// TwinCAT 3 PLC project CX5240
// ProgramVersion: 3.1.4026.13
// CompilerDefines: VISU_USEPROPERTYINFO
// libraries:
//   CmpBitmapPool, * (System)
//   Tc2_Standard, * (Beckhoff Automation GmbH)
//   Tc2_System, * (Beckhoff Automation GmbH)
//   Tc3_Module, * (Beckhoff Automation GmbH)
//   VisuDialogs, * (System)
//   VisuSymbols,3.5.10.0,System
// project tree:
//   Enums/ E_Status.TcDUT (not stored)
//   Function Blocks/ FB_AnalogInputScaling.TcPOU (not stored), FB_DisplacementControl.TcPOU (not stored), FB_Encoder.TcPOU (not stored), FB_Integrator.TcPOU (not stored), FB_Joystick.TcPOU (not stored), FB_JoystickInputScaling.TcPOU (not stored), FB_DisplacementValveOutput.TcPOU (not stored), FB_StartPos.TcPOU (not stored), FB_YokeInputScaling.TcPOU (not stored), FB_ValveOutput.TcPOU (not stored)
//   / GlobalTextList.TcGTLO, HMI.TcVIS, PlcTask.TcTTO (not stored), Visualization Manager.TcVMO (not stored)
//   GVLs/ G_IO.TcGVL, G_Parameters.TcGVL, G_Sensors.TcGVL (not stored), HMI.TcGVL
//   POUs/ MAIN.TcPOU (not stored), P_Inputs.TcPOU, P_MotionControl.TcPOU, P_Outputs.TcPOU (not stored)
//   Struct/ ST_AnalogInputScaling.TcDUT (not stored), ST_JoystickInputScaling.TcDUT (not stored), ST_YokeInputScaling.TcDUT (not stored), ST_Parameters.TcDUT (not stored), ST_ValveDeadBand.TcDUT (not stored), ST_ValveOutput.TcDUT (not stored)
// real-time tasks:
//   TASK PlcTask: cycle T#1ms, priority 20, ADS port 350
// I/O:
//   DEVICE Device 1 (EtherCAT), AmsNetId 128.39.200.126.2.1
//     Term 1 (EK1200) [EK1200-5000 EtherCAT Power supply (2A E-Bus)]
//       Term 2 (EL1859) [EL1859 8Ch. Dig. Input 24V, 3ms, 8Ch. Dig. Output 24V, 0.5A]
//       Term 3 (EL3174) [EL3174 4Ch. Ana. Input +/-10V Diff., +/-20mA SingleEnded, 16 Bit]
//       Term 4 (EL4032) [EL4032 2Ch. Ana. Output +/-10V, 12bit]
//       Term 7 (EL3204) [EL3204 4Ch. Ana. Input PT100 (RTD)]
//       Term 8 (EK1110) [EK1110 EtherCAT extension]
//     Term 14 (EK1818) [EK1818 EtherCAT IO-Coupler  (1A E-Bus, 8 Ch. Dig. In, 3ms, 4 Ch. Dig. Out 24V, 0,5A)]
//       Term 10 (EL1008) [EL1008 8Ch. Dig. Input 24V, 3ms]
//       Term 11 (EL3174) [EL3174 4Ch. Ana. Input +/-10V Diff., +/-20mA SingleEnded, 16 Bit]
//       Term 12 (EL3068) [EL3068 8Ch. Ana. Input 0-10V]
//       Term 5 (EL4032) [EL4032 2Ch. Ana. Output +/-10V, 12bit]
//       Term 6 (EL4122) [EL4122 2Ch. Ana. Output  4-20mA, 16bit]
//       Term 17 (EL9011) [EL9011 End Terminal]
//     Box 13 (Fraba EtherCAT) [Absolute Rotary Encoder IXARC V01.05]
// variable links:
//   CX5240/CX5240 Instance <-> Device 1 (EtherCAT)/Term 1 (EK1200)/Term 2 (EL1859)
//     PlcTask Inputs/G_IO.bTestNew <-> Channel 1/Input
//     PlcTask Outputs/G_IO.OutTestNew <-> Channel 9/Output
//   CX5240/CX5240 Instance <-> Device 1 (EtherCAT)/Term 1 (EK1200)/Term 3 (EL3174)
//     PlcTask Inputs/G_IO.nTestNew <-> AI Standard Channel 1/Value
//   CX5240/CX5240 Instance <-> Device 1 (EtherCAT)/Term 14 (EK1818)
//     PlcTask Inputs/G_IO.bEmgOk <-> Channel 1/Input
//     PlcTask Outputs/G_IO.bEnablePCDV <-> Channel 10/Output
//     PlcTask Outputs/G_IO.bOpenBrakes <-> Channel 9/Output
//     PlcTask Outputs/G_IO.bWinchValveEnable <-> Channel 11/Output
//   CX5240/CX5240 Instance <-> Device 1 (EtherCAT)/Term 14 (EK1818)/Term 10 (EL1008)
//     PlcTask Inputs/G_IO.bAutoSwtich <-> Channel 3/Input
//     PlcTask Inputs/G_IO.bDisplacementEnable <-> Channel 7/Input
//     PlcTask Inputs/G_IO.bManualSwtich <-> Channel 1/Input
//     PlcTask Inputs/G_IO.bOffSwtich <-> Channel 2/Input
//     PlcTask Inputs/G_IO.bStartButton <-> Channel 4/Input
//     PlcTask Inputs/G_IO.bStopButton <-> Channel 5/Input
//     PlcTask Inputs/G_IO.bWinchEnable <-> Channel 6/Input
//   CX5240/CX5240 Instance <-> Device 1 (EtherCAT)/Term 14 (EK1818)/Term 11 (EL3174)
//     PlcTask Inputs/G_IO.fPDCVMonitor <-> AI Standard Channel 1/Value
//     PlcTask Inputs/G_IO.fYoke <-> AI Standard Channel 4/Value
//     PlcTask Inputs/G_IO.nMoogMonitor <-> AI Standard Channel 2/Value
//   CX5240/CX5240 Instance <-> Device 1 (EtherCAT)/Term 14 (EK1818)/Term 12 (EL3068)
//     PlcTask Inputs/G_IO.fJoyXraw <-> AI Standard Channel 6/Value
//     PlcTask Inputs/G_IO.fJoyYraw <-> AI Standard Channel 7/Value
//     PlcTask Inputs/G_IO.fJoyZraw <-> AI Standard Channel 8/Value
//     PlcTask Inputs/G_IO.fPressureReturn <-> AI Standard Channel 3/Value
//     PlcTask Inputs/G_IO.fPressureSupply <-> AI Standard Channel 2/Value
//     PlcTask Inputs/G_IO.fPressureWinchA <-> AI Standard Channel 1/Value
//     PlcTask Inputs/G_IO.fPressureWinchB <-> AI Standard Channel 4/Value
//   CX5240/CX5240 Instance <-> Device 1 (EtherCAT)/Term 14 (EK1818)/Term 5 (EL4032)
//     PlcTask Outputs/G_IO.fWinchPDCVOut <-> AO Outputs Channel 1/Analog output
//   CX5240/CX5240 Instance <-> Device 1 (EtherCAT)/Term 14 (EK1818)/Term 6 (EL4122)
//     PlcTask Outputs/G_IO.fWinchValveOut <-> Channel 1/Output

// ---- GVLs/G_IO.TcGVL
{attribute 'qualified_only'}
VAR_GLOBAL
	// Digital Inputs
	bEmgOk 			     AT %I* : BOOL; 
	bStartButton 	     AT %I* : BOOL;
	bStopButton 	     AT %I* : BOOL; 
	bOffSwtich		     AT %I* : BOOL;  
	bManualSwtich	     AT %I* : BOOL; 
	bAutoSwtich			 AT %I* : BOOL; 
	bWinchEnable 		 AT %I* : BOOL; 
	bDisplacementEnable  AT %I* : BOOL;
	
	// Analog Intputs
	fJoyXraw 			 AT %I* : INT; 
	fJoyYraw			 AT %I* : INT; 
	fJoyZraw 			 AT %I* : INT; 
	fPDCVMonitor		 AT %I* : INT; 
	nMoogMonitor		 AT %I* : INT; 
	fYoke				 AT %I* : INT; 
	fPressureWinchA 	 AT %I* : INT; 
	fPressureWinchB 	 AT %I* : INT; 
	fPressureSupply 	 AT %I* : INT; 
	fPressureReturn 	 AT %I* : INT; 
	nWinchEncoderValue	 AT %I* : UDINT; 
	
	// Digital Outputs
	bOpenBrakes 		 AT %Q* : BOOL; 
	bEnablePCDV 		 AT %Q* : BOOL; 
	bWinchValveEnable 	 AT %Q* : BOOL; 
	
	// Analog Outputs
	fWinchPDCVOut 		 AT %Q* : INT := 10000; 
	fWinchValveOut 		 AT %Q* : INT := 16383; 
	
	// New Test
	bTestNew AT %I* : BOOL;
	nTestNew AT %I* : INT;
	
END_VAR

// ---- GVLs/G_Parameters.TcGVL
{attribute 'qualified_only'}
VAR_GLOBAL
stParam : ST_Parameters;
END_VAR

// ---- GVLs/HMI.TcGVL
{attribute 'qualified_only'}
VAR_GLOBAL
	bEndStopOverride : BOOL; 
	fTest			 : LREAL;
END_VAR

// ---- POUs/P_Inputs.TcPOU
PROGRAM P_Inputs
VAR
	fbJoystickWinch 				: FB_JoystickInputScaling;
	fbJoystickRot 					: FB_JoystickInputScaling;
	fbYokeInputScaling 				: FB_YokeInputScaling;
	fbWinchPosition 				: FB_Encoder;
	fbPressureSupply 				: FB_AnalogInputScaling;
	fbPressureReturn 				: FB_AnalogInputScaling;
	fbPressureWinch_A_Input 		: FB_AnalogInputScaling;
	fbPressureWinch_B_Output		: FB_AnalogInputScaling;
END_VAR

fbJoystickWinch(
	bEnable := G_IO.bManualSwtich OR G_IO.bAutoSwtich,
	nRawInput := G_IO.fJoyYraw,
	stJoystickInputScaling := G_Parameters.stParam.stJoystickInputScalingY,
	fNormalizedOutput => G_Sensors.fJoystickNormalizedY
);

fbJoystickRot(
	bEnable := G_IO.bManualSwtich,
	nRawInput := G_IO.fJoyZraw,
	stJoystickInputScaling := G_Parameters.stParam.stJoystickInputScalingZ,
	fNormalizedOutput => G_Sensors.fJoystickNormalizedZ
);

fbYokeInputScaling(
	bEnable := G_IO.bManualSwtich,
	nRawInput := G_IO.fYoke,
	stYokeInputScaling := G_Parameters.stParam.stYokeInputScaling,
	fNormalizedOutput => G_Sensors.fYokeNormalizedFeedback
);

fbWinchPosition (
	nRawInput := G_IO.nWinchEncoderValue, 
	fEncoderOffset := G_Parameters.stParam.fWinchEncoderOffset,
	fPosition => G_Sensors.fWinchEncoderPosition
);

fbPressureSupply(
	nRawInput := G_IO.fPressureSupply,
	stAnalogInputScaling := G_Parameters.stParam.stPressureSensorScaling400bar,
	fOutput => G_Sensors.fPressureSupply
);

fbPressureReturn(
	nRawInput := G_IO.fPressureReturn,
	stAnalogInputScaling := G_Parameters.stParam.stPressureSensorScaling40bar,
	fOutput => G_Sensors.fPressureReturn
);

fbPressureWinch_A_Input(
	nRawInput := G_IO.fPressureWinchA,
	stAnalogInputScaling := G_Parameters.stParam.stPressureSensorScaling400bar,
	fOutput => G_Sensors.fPressureWinchA
);

fbPressureWinch_B_Output(
	nRawInput := G_IO.fPressureCylinderA,
	stAnalogInputScaling := G_Parameters.stParam.stPressureSensorScaling400bar,
	fOutput => G_Sensors.fPressureWinchB
);

G_Sensors.fDeltaPMotor := (G_Sensors.fPressureWinchB - G_Sensors.fPressureWinchA);

END_PROGRAM

// ---- POUs/P_MotionControl.TcPOU
PROGRAM P_MotionControl
VAR
	fbJoystick 				: FB_Joystick;
	fbGetStartPos 			: FB_StartPos;
	fbWinchVelIntegrator 	: FB_Integrator;
	fWinchVelRef 			: LREAL;
	fWinchPosRef 			: LREAL;
	fWinchPos 				: LREAL;
	fInitialWinchPos 		: LREAL;
	bWinchVelIntegratorOn	: BOOL := TRUE; 
	bAutoEnable 			: BOOL;
	bManualEnable 			: BOOL;
	fWinchPosRefManual 		: LREAL;
	fWinchVelRefManual 		: LREAL;
	fWinchVelRefAuto 		: LREAL;
	fbJoyTest 				: FB_Joystick;
END_VAR

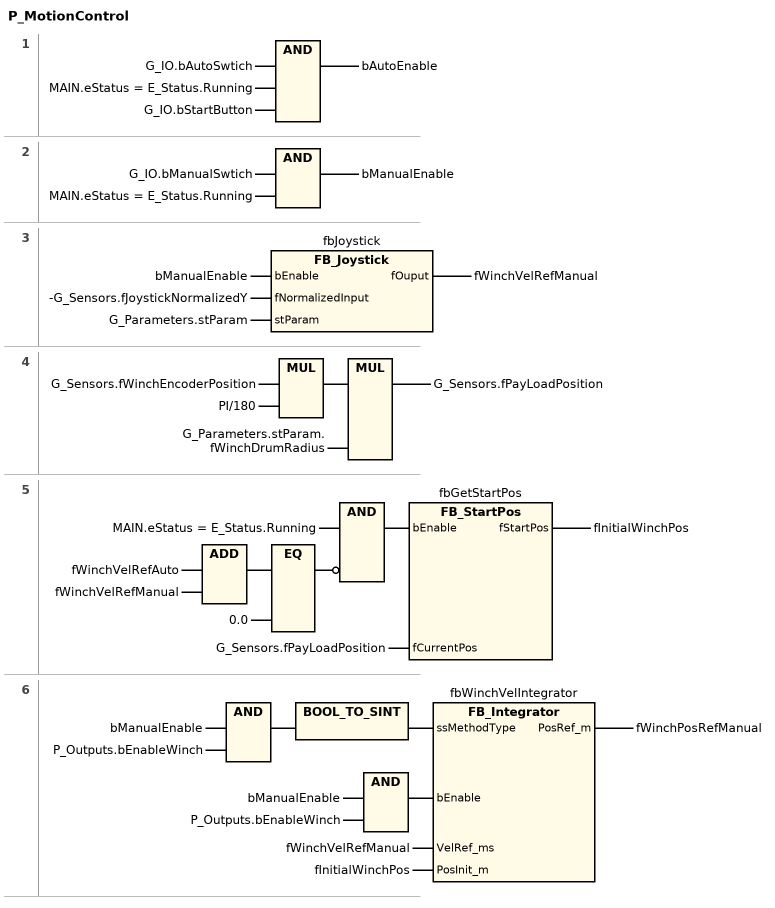
// NETWORK 1
bAutoEnable := G_IO.bAutoSwtich AND (MAIN.eStatus = E_Status.Running) AND G_IO.bStartButton;

// NETWORK 2
bManualEnable := G_IO.bManualSwtich AND (MAIN.eStatus = E_Status.Running);

// NETWORK 3
fbJoystick(
    bEnable := bManualEnable,
    fNormalizedInput := -G_Sensors.fJoystickNormalizedY,
    stParam := G_Parameters.stParam); // FB_Joystick
fWinchVelRefManual := fbJoystick.fOuput;

// NETWORK 4
G_Sensors.fPayLoadPosition := (G_Sensors.fWinchEncoderPosition * (PI/180)) * G_Parameters.stParam.fWinchDrumRadius;

// NETWORK 5
fbGetStartPos(bEnable := (MAIN.eStatus = E_Status.Running) AND NOT (fWinchVelRefAuto + fWinchVelRefManual = 0.0), fCurrentPos := G_Sensors.fPayLoadPosition); // FB_StartPos
fInitialWinchPos := fbGetStartPos.fStartPos;

// NETWORK 6
fbWinchVelIntegrator(
    ssMethodType := BOOL_TO_SINT(bManualEnable AND P_Outputs.bEnableWinch),
    bEnable := bManualEnable AND P_Outputs.bEnableWinch,
    VelRef_ms := fWinchVelRefManual,
    PosInit_m := fInitialWinchPos); // FB_Integrator
fWinchPosRefManual := fbWinchVelIntegrator.PosRef_m;

END_PROGRAM

// ---- GlobalTextList.TcGTLO
TEXTLIST GlobalTextList
  455 = '%2.1f'
  509 = '%2.2f'
  108 = '%f'
  308 = '%i'
  805 = '%I'
  528 = "'amplitude"
  341 = 'A'
  810 = 'Actvting Log P'
  221 = 'Actvting Log Plat'
  505 = 'Actvting Log Pos'
  560 = 'Amplitud'
  159 = 'Amplitude'
  639 = 'bar'
  175 = 'Controlelr'
  786 = 'Controller'
  847 = 'D'
  489 = 'END STOP OVERRIDE'
  897 = 'END STOP OVERRIDE '
  616 = 'EndStop Override'
  141 = 'GO TO SETTINGS'
  499 = 'I'
  490 = 'Main'
  911 = 'Main Screen'
  508 = 'Motion Control'
  934 = 'MOTION LIMIT'
  673 = 'Motion Limit'
  176 = 'MOTION LIMIT: OFF'
  449 = 'MOTION LIMITATION'
  802 = 'MOTION LIMITATION: OFF'
  69 = 'Neg End Stop'
  444 = 'Neg EndStop'
  896 = 'OVERRIDE'
  993 = 'P'
  312 = 'PA bar'
  288 = 'PA Winch bar'
  641 = 'PB bar'
  622 = 'PI COntroler'
  326 = 'PI Controler'
  878 = 'PI Displacement Control'
  623 = 'PI Gain DC'
  962 = 'PI Gain P'
  177 = 'PI Gain SC'
  28 = 'PI Primary Control'
  144 = 'PI Secondary Control'
  68 = 'PID'
  907 = 'PID Contoler'
  714 = 'PID Controller'
  706 = 'Pos End Stop'
  398 = 'Pos EndStop'
  309 = 'Position Logging'
  953 = 'Screen'
  358 = 'Secondary Control'
  699 = 'Secondry'
  663 = 'Secondry  swicher Primery'
  725 = 'Secondry Control'
  395 = 'Secondry Ish'
  17 = 'Secondry Swicher Primery'
  238 = 'Setings'
  169 = 'Settings'
  590 = 'Sin AmplitudContoler'
  156 = 'Sin TimeP Contoler'
  94 = 'Sin Wave'
  613 = 'Sin Wave Contoler'
  420 = 'Sine Motion Off/On'
  636 = 'Sine Wave'
  818 = 'Start Mual'
  898 = 'Time'
  26 = 'Time P'
  140 = 'Time Periode [s]'
  844 = 'TimeP'
  826 = 'TimePTime'
  402 = 'to Main'
  655 = 'Togel Swich Motion Control'
  469 = 'TURN ON IN SETTINGS'
  191 = 'Visualisation'
  345 = 'Visualiztion'
  718 = 'WARNING'
  113 = 'Warning ON'
  628 = 'Wave Amplitude [m]'
  592 = 'Working Progres'
  500 = 'XXX'
END_TEXTLIST

// ---- HMI.TcVIS
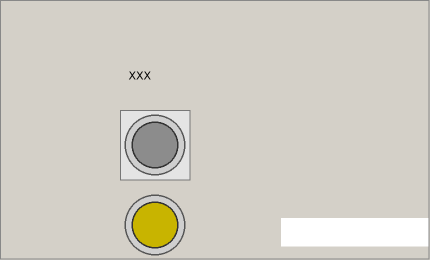
VISUALIZATION HMI  // 430x260
    PushSwitch (120,110 70x70), variable: HMI.bEndStopOverride, behaviour: TOGGLE, style: Switch-PushSwitch-Gray
    Lamp1 (120,190 70x70), variable: G_IO.bManualSwtich, style: Lamp-Lamp1-Yellow
    Label (65,61 150x30), "XXX"
    Textfield (280,217 150x30), text variable: HMI.fTest
END_VISUALIZATION
